{attribute 'linkalways'} 
{attribute 'no_explicit_call' := 'This FB is a CLASS and must be accessed using methods or properties'}
{attribute 'enable_dynamic_creation'}
FUNCTION_BLOCK Node_F_VN_FillContainerExp_DINT EXTENDS VisionNode
VAR
    ipContainer : _ITcVnContainer;
    nValue : _DINT(0);
    nStartIdx : _ULINT(0);
    nCount : _ULINT(0);
    hrPrev : _HRESULT(S_OK);
    hresult : _HRESULT(S_OK);
END_VAR

METHOD PUBLIC  Clone : I_Node
VAR
    pNode : POINTER TO Node_F_VN_FillContainerExp_DINT;
END_VAR
pNode := __NEW(Node_F_VN_FillContainerExp_DINT);
Clone := pNode^;
END_METHOD

METHOD FB_init : BOOL
VAR_INPUT
    bInitRetains : BOOL; // if TRUE, the retain variables are initialized (warm start / cold start)
    bInCopyCode : BOOL;  // if TRUE, the instance afterwards gets moved into the copy code (online change)
END_VAR
AddInput('ipContainer', ipContainer);
AddParameter('nValue', nValue);
AddParameter('nStartIdx', nStartIdx);
AddParameter('nCount', nCount);
AddInput('hrPrev', hrPrev);
AddOutput('ipContainer', ipContainer);
AddOutput('hresult',hresult);
END_METHOD

METHOD PROTECTED OnExecute
hresult.Value := F_VN_FillContainerExp_DINT(
    ipContainer := ipContainer.Value,
    nValue := nValue.Value,
    nStartIdx := nStartIdx.Value,
    nCount := nCount.Value,
    hrPrev:= hrPrev.Value);
END_METHOD

METHOD PUBLIC PreExecutionCheck
VAR_INPUT
    Check : I_PreExecutionChecks;
END_VAR
Check.IsTrue(ipContainer.IsValid, 'ipContainer must be a valid container');
Check.IsTrue(ipContainer.IsType(TC_GLOBAL_CONST_LIST.ContainerType_Vector_DINT), 'ipContainer contains incorrect type');
END_METHOD

END_FUNCTION_BLOCK

(* stored: Version 1.1.0.1, ProductVersion 3.1.4026.13
   POU Node_F_VN_FillContainerExp_DINT: Id {2290eaa5-4b14-4348-b06c-572f5257cc74}, SpecialFunc None
   Folder Constructor: Id {0e5cc048-fccf-4da5-90ea-50dd9e735e46}
   Method Clone: Id {1f088f9a-85cc-442d-8f7b-86d7154fe21c}
   Method FB_init: Id {16083af0-b9b7-404d-93ca-4b418772aeb3}
   Method OnExecute: Id {cca3e0f3-39ca-4f17-bba1-561b09f4b6b4}
   Method PreExecutionCheck: Id {f52cbbce-94dd-4952-a863-df4f31e18109} *)
